PROGRAM TP_and_TON_For_timeout
VAR
	TP_1_trigger: BOOL;
	TP_1: TP;
	Trig_TON_1: BOOL;
	TON_1: TON;
	TP_2_trigger: BOOL;
	TP_2: TP;
	Trig_TON_2: BOOL;
	TON_2: TON;
END_VAR

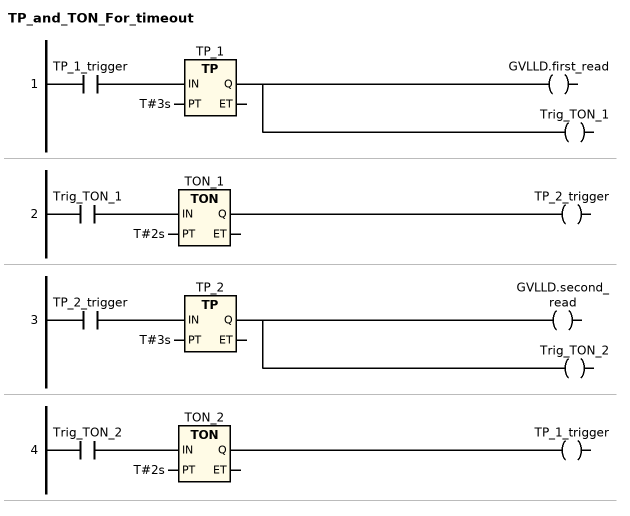
// NETWORK 1
TP_1(IN := TP_1_trigger, PT := T#3s); // TP
GVLLD.first_read := TP_1.Q;
Trig_TON_1 := TP_1.Q;

// NETWORK 2
TON_1(IN := Trig_TON_1, PT := T#2s); // TON
TP_2_trigger := TON_1.Q;

// NETWORK 3
TP_2(IN := TP_2_trigger, PT := T#3s); // TP
GVLLD.second_read := TP_2.Q;
Trig_TON_2 := TP_2.Q;

// NETWORK 4
TON_2(IN := Trig_TON_2, PT := T#2s); // TON
TP_1_trigger := TON_2.Q;

END_PROGRAM

(* stored: Version 1.1.0.1, ProductVersion 3.1.4024.12
   POU TP_and_TON_For_timeout: Id {94d90764-1941-4f16-b049-067b4ca5d2dc}, SpecialFunc None *)
